FUNCTION Mapping_ModbusWriteRegisters : bool
VAR_INPUT
	//Modbus_Structure : POINTER TO MOdbusWrite_NRG;
	Modbus_Structure : POINTER TO ModbusWrite;
	FromSLC : POINTER TO EtherCAT_Inputs;
END_VAR
VAR
	wAutoManCtl: INT;
END_VAR

//Commands
	//State machine operation
		Modbus_Structure^.CmdOpMode := REAL_TO_INT(FromSLC^.Command);
	//Power Reference
		//Modbus_Structure^.Pset := (FromSLC^.ActivePowerReference);
		//Modbus_Structure^.Qset := (FromSLC^.ReactivePowerReference);

//GlobalVar.ModWrite.SLC_Debugger := FromSLC^.Commands;

END_FUNCTION

(* stored: Version 1.1.0.1, ProductVersion 3.1.4024.2
   POU Mapping_ModbusWriteRegisters: Id {4fcede58-d6bc-46b0-a7db-ae8676c0e79a}, SpecialFunc None *)
